// TwinCAT 3 PLC project Untitled1
// ProgramVersion: 3.1.4024.0
// libraries:
//   SPT Base Types, * (Beckhoff Automation LLC)
//   SPT Components, * (Beckhoff Automation LLC)
//   SPT Motion Control, * (Beckhoff Automation LLC)
//   Tc2_MC2, * (Beckhoff Automation GmbH)
//   Tc2_Standard, * (Beckhoff Automation GmbH)
//   Tc2_System, * (Beckhoff Automation GmbH)
//   Tc3_Module, * (Beckhoff Automation GmbH)
//   Tc3_PackML_V2, * (Beckhoff Automation GmbH)
// project tree:
//   Machine/EquipmentModules/ FB_DrawAxis.TcPOU, FB_Unwind.TcPOU, FB_VM.TcPOU (not stored)
//   Machine/MachineModule/ FB_Machine.TcPOU
//   / PlcTask.TcTTO (not stored)
//   POUs/ MAIN.TcPOU

// ---- Machine/EquipmentModules/FB_DrawAxis.TcPOU
{attribute 'no_explicit_call' := 'This FB is a CLASS and must be accessed using methods or properties'}
FUNCTION_BLOCK FB_DrawAxis EXTENDS FB_PackML_BaseModule
VAR
	Axis	  : FB_Component_BasicSlaveAxis := (Name := 'Draw Axis');
	MasterRef : REFERENCE TO AXIS_REF;
END_VAR

METHOD PROTECTED Aborting
// Mode is ignored
CASE SequenceState OF
	0:
		NoStateTasksToComplete := FALSE;
		SequenceState		   := SequenceState + 10;

	10: // Stop Axis
		Axis.Override := 100;
		Axis.Stop(); // This will also GearOut by default
		IF Axis.Stopped THEN
			SequenceState := SequenceState + 10;
		END_IF

	20: // Disable Axis
		Axis.Disable();
		IF NOT Axis.Enabled THEN
			StateTasksComplete := TRUE;
		END_IF
END_CASE

SUPER^.Aborting();
END_METHOD

PROPERTY AxisRef : REFERENCE TO AXIS_REF
GET
AxisRef REF= Axis.Axis;
END_GET
END_PROPERTY

METHOD PROTECTED Completing
CASE _CurrentMode OF
	ePMLUnitMode_Production:
		CASE SequenceState OF
			0:
				NoStateTasksToComplete := FALSE;
				SequenceState		   := SequenceState + 10;

			10: // Wait for Master Axis to Stop and GearOut, or Stop
				IF Axis.InGear AND Axis.Stopped THEN
					Axis.GearOut();
				ELSIF NOT Axis.InGear THEN
					Axis.Stop();
				END_IF

				IF Axis.Stopped THEN
					StateTasksComplete := TRUE;
				END_IF
		END_CASE
END_CASE

SUPER^.Completing();
END_METHOD

METHOD PUBLIC CyclicLogic
IF NOT _InitComplete THEN
	_InitComplete := Initialize();
	RETURN;
END_IF

SUPER^.CyclicLogic();
END_METHOD

METHOD PROTECTED Initialize : BOOL;
VAR
	i : UDINT;
END_VAR
Initialize := FALSE;
CASE DescendantSequenceState OF
	0: // Register Components
		RegisterComponent(Axis);

		// Set Config
		_LogModeChanges			:= FALSE;
		_LogStateChanges		:= FALSE;
		DescendantSequenceState := DescendantSequenceState + 10;

	10: // Copy Mode names
		FOR i := 1 TO 10 DO
			ModeNames[i] := F_UnitModeToString(UDINT_TO_DINT(i));
		END_FOR

		DescendantSequenceState := DescendantSequenceState + 10;

	20:
		IF SUPER^.Initialize() THEN
			DescendantSequenceState := DescendantSequenceState + 10;
		END_IF

	30:
		Initialize := TRUE;
END_CASE
END_METHOD

PROPERTY MasterAxisRef : REFERENCE TO AXIS_REF
SET
MasterRef REF= MasterAxisRef;
END_SET
END_PROPERTY

METHOD PROTECTED Starting
CASE _CommandedMode OF
	ePMLProtUnitMode_Production:
		CASE SequenceState OF
			0:
				NoStateTasksToComplete := FALSE;
				SequenceState		   := SequenceState + 10;

			10: // Enable Axis
				Axis.Enable();
				IF Axis.Enabled THEN
					SequenceState := SequenceState + 10;
				END_IF

			20: // Set reference to Master and Couple Axes
				Axis.Master1 REF= MasterRef;
				Axis.GearIn();
				IF Axis.InGear THEN
					StateTasksComplete := TRUE;
				END_IF
		END_CASE
END_CASE

SUPER^.Starting();
END_METHOD

METHOD PROTECTED Stopping
CASE _CurrentMode OF
	ePMLUnitMode_Production:
		CASE SequenceState OF
			0:
				NoStateTasksToComplete := FALSE;
				SequenceState		   := SequenceState + 10;

			10: // Stop Axis
				Axis.Override := 100;
				Axis.Stop(); // This will also GearOut by default
				IF Axis.Stopped THEN
					StateTasksComplete := TRUE;
				END_IF
		END_CASE
END_CASE

SUPER^.Stopping();
END_METHOD

END_FUNCTION_BLOCK

// ---- Machine/EquipmentModules/FB_Unwind.TcPOU
{attribute 'no_explicit_call' := 'This FB is a CLASS and must be accessed using methods or properties'}
FUNCTION_BLOCK FB_Unwind EXTENDS FB_PackML_BaseModule
VAR
	Axis	  : FB_Component_BasicSlaveAxis := (Name := 'Unwind Axis');
	MasterRef : REFERENCE TO AXIS_REF;
END_VAR

METHOD PROTECTED Aborting
// Mode is ignored
CASE SequenceState OF
	0:
		NoStateTasksToComplete := FALSE;
		SequenceState		   := SequenceState + 10;

	10: // Stop Axis
		Axis.Override := 100;
		Axis.Stop(); // This will also GearOut
		IF Axis.Stopped THEN
			SequenceState := SequenceState + 10;
		END_IF

	20: // Disable Axis
		Axis.Disable();
		IF NOT Axis.Enabled THEN
			StateTasksComplete := TRUE;
		END_IF
END_CASE

SUPER^.Aborting();
END_METHOD

PROPERTY AxisRef : REFERENCE TO AXIS_REF
GET
AxisRef REF= Axis.Axis;
END_GET
END_PROPERTY

METHOD PROTECTED Completing
CASE _CurrentMode OF
	ePMLUnitMode_Production:
		CASE SequenceState OF
			0:
				NoStateTasksToComplete := FALSE;
				SequenceState		   := SequenceState + 10;

			10: // Wait for Master Axis to Stop and GearOut, or Stop
				IF Axis.InGear AND Axis.Stopped THEN
					Axis.GearOut();
				ELSIF NOT Axis.InGear THEN
					Axis.Stop();
				END_IF

				IF Axis.Stopped THEN
					StateTasksComplete := TRUE;
				END_IF
		END_CASE
END_CASE

SUPER^.Completing();
END_METHOD

METHOD PUBLIC CyclicLogic
IF NOT _InitComplete THEN
	_InitComplete := Initialize();
	RETURN;
END_IF

SUPER^.CyclicLogic();
END_METHOD

METHOD PROTECTED Initialize : BOOL;
VAR
	i : UDINT;
END_VAR
Initialize := FALSE;
CASE DescendantSequenceState OF
	0: // Register Components
		RegisterComponent(Axis);

		// Set Config
		_LogModeChanges			:= FALSE;
		_LogStateChanges		:= FALSE;
		DescendantSequenceState := DescendantSequenceState + 10;

	10:
		// Copy Mode names
		FOR i := 1 TO 10 DO
			ModeNames[i] := F_UnitModeToString(UDINT_TO_INT(i));
		END_FOR

		DescendantSequenceState := DescendantSequenceState + 10;

	20:
		IF SUPER^.Initialize() THEN
			DescendantSequenceState := DescendantSequenceState + 10;
		END_IF

	30:
		Initialize := TRUE;
END_CASE
END_METHOD

PROPERTY MasterAxisRef : REFERENCE TO AXIS_REF
SET
MasterRef REF= MasterAxisRef;
END_SET
END_PROPERTY

METHOD PROTECTED Starting
CASE _CommandedMode OF
	ePMLProtUnitMode_Production:
		CASE SequenceState OF
			0:
				NoStateTasksToComplete := FALSE;
				SequenceState		   := SequenceState + 10;

			10: // Enable Axis
				Axis.Enable();
				IF Axis.Enabled THEN
					SequenceState := SequenceState + 10;
				END_IF

			20: // Set reference to Master and Couple Axes
				Axis.Master1	  REF= MasterRef;
				Axis.RatioMaster1 := 0.5; // Can be set at anytime and changed while in motion
				Axis.GearIn();
				IF Axis.InGear THEN
					StateTasksComplete := TRUE;
				END_IF
		END_CASE
END_CASE

SUPER^.Starting();
END_METHOD

METHOD PROTECTED Stopping
CASE _CurrentMode OF
	ePMLUnitMode_Production:
		CASE SequenceState OF
			0:
				NoStateTasksToComplete := FALSE;
				SequenceState		   := SequenceState + 10;

			10: // Stop Axis
				Axis.Override := 100;
				Axis.Stop(); // This will also GearOut
				IF Axis.Stopped THEN
					StateTasksComplete := TRUE;
				END_IF
		END_CASE
END_CASE

SUPER^.Stopping();
END_METHOD

END_FUNCTION_BLOCK

// ---- Machine/MachineModule/FB_Machine.TcPOU
{attribute 'no_explicit_call' := 'This FB is a CLASS and must be accessed using methods or properties'}
FUNCTION_BLOCK FB_Machine EXTENDS FB_PackML_BaseModule
VAR
	VirtualMaster : FB_VM		:= (Name := 'Virtual Master');
	Unwind		  : FB_Unwind	:= (Name := 'Unwind EM');
	Draw		  : FB_DrawAxis := (Name := 'Draw EM');
END_VAR

METHOD PUBLIC CyclicLogic
IF NOT _InitComplete THEN
	_InitComplete := Initialize();
	RETURN;
END_IF

SUPER^.CyclicLogic();
END_METHOD

METHOD PROTECTED Initialize : BOOL;
VAR
	i : UDINT;
END_VAR
Initialize := FALSE;
CASE DescendantSequenceState OF
	0: // Register Submodules
		RegisterSubmodule(VirtualMaster);
		RegisterSubmodule(Unwind);
		RegisterSubmodule(Draw);

		// Register Components

		// Set Config
		_LogModeChanges			:= FALSE;
		_LogStateChanges		:= FALSE;
		DescendantSequenceState := DescendantSequenceState + 10;

	10: // Setup Custom modes here
		DescendantSequenceState := DescendantSequenceState + 10;

	20: // Copy Mode names
		FOR i := 1 TO 10 DO
			ModeNames[i] := F_UnitModeToString(UDINT_TO_DINT(i));
		END_FOR

		DescendantSequenceState := DescendantSequenceState + 10;

	30: // Default recipe values parameters entered here
		Unwind.MasterAxisRef	REF= VirtualMaster.AxisRef;
		Draw.MasterAxisRef		REF= VirtualMaster.AxisRef;
		DescendantSequenceState := DescendantSequenceState + 10;

	40:
		IF SUPER^.Initialize() THEN
			Initialize := TRUE;
		END_IF
END_CASE
END_METHOD

END_FUNCTION_BLOCK

// ---- POUs/MAIN.TcPOU
PROGRAM MAIN
VAR
	Machine	  : FB_Machine;
	nextState : BOOL;
	abort	  : BOOL;
	stop	  : BOOL;
	curState  : E_PMLState;
END_VAR

// All sample code provided by Beckhoff Automation LLC are for illustrative purposes only and are provided “as is” and without any warranties, express or implied. Actual implementations in applications will vary significantly. Beckhoff Automation LLC shall have no liability for, and does not waive any rights in relation to, any code samples that it provides or the use of such code samples for any purpose.

(*
This sample displays how an axis component of an EM can be coupled to the axis component of another EM.
The Unwind Axis makes use of a Gear Ratio in its Coupling - see FB_Unwind.Starting step 20.
The configuration for setting the reference to the Master Axis is done in FB_Machine.Initialize step 20.

This code is not a full implementation as there is no use of MC_Reset or other needed code for actual machine use.
There is no code to move the master axis, but it can be jogged from the NC for testing.

*)
Machine.CyclicLogic();

// For display purposes as local variable
curState := Machine.CurrentState;

// Toggle to move to next state
IF nextState THEN
	nextState := FALSE;
	CASE Machine.CurrentState OF
		ePMLState_Aborted:
			Machine.ChangeState(State := ePMLCommand_Clear);

		ePMLState_Stopped, ePMLState_Complete:
			Machine.ChangeState(State := ePMLCommand_Reset);

		ePMLState_Idle:
			Machine.ChangeState(State := ePMLCommand_Start);

		ePMLState_Execute:
			Machine.ChangeState(State := ePMLCommand_Complete);
	END_CASE
END_IF

IF abort THEN
	abort := FALSE;
	Machine.ChangeState(State := ePMLCommand_Abort);
END_IF

IF stop THEN
	stop := FALSE;
	Machine.ChangeState(State := ePMLCommand_Stop);
END_IF

END_PROGRAM
